(* PLC project My_First_Project, Unknown Unnamed 1 *)
(* stored: creationDateTime 2020-02-11T22:16:33, modificationDateTime 2020-02-11T22:24:10 *)

PROGRAM My_First_Program
  VAR
    PB1 AT %IX0.0 : BOOL;
    PB2 AT %IX0.1 : BOOL;
    LAMP AT %QX0.0 : BOOL;
  END_VAR

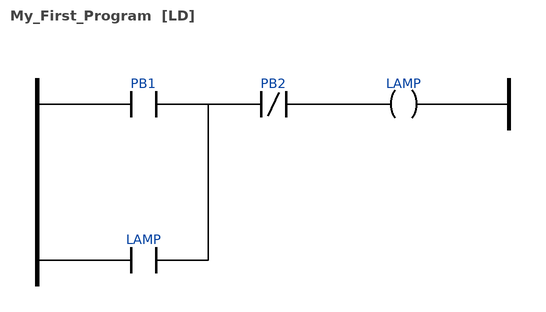
(* LD diagram, written out as Structured Text *)
LAMP := (PB1 OR LAMP) AND NOT PB2;
END_PROGRAM

CONFIGURATION Config0
  RESOURCE Res0 ON PLC
    TASK task0(INTERVAL := T#20ms, PRIORITY := 0);
    PROGRAM instance0 WITH task0 : My_First_Program;
  END_RESOURCE
END_CONFIGURATION
